// SIMATIC S7-200 project (STEP 7-Micro/WIN), CPU 224 CN REL 02.02

ORGANIZATION_BLOCK 主程序:OB1
TITLE=程序注释
BEGIN
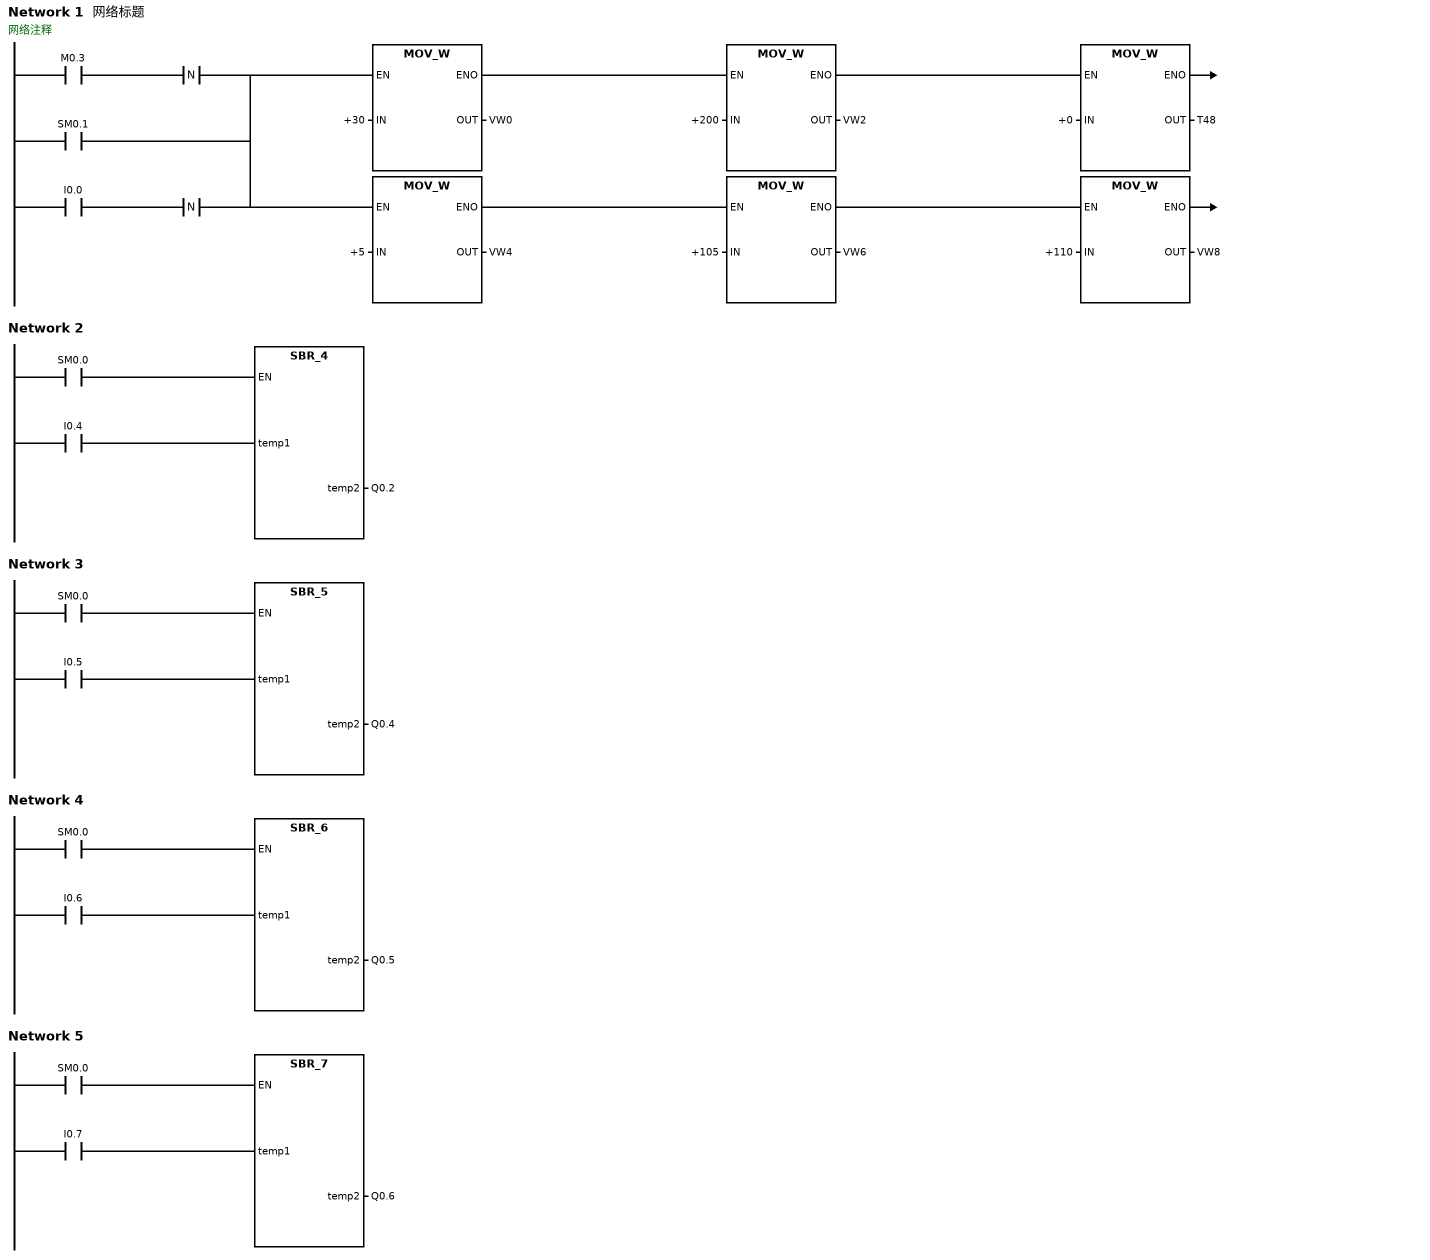
Network 1 // 网络标题
// 网络注释
LD     M0.3
ED
O      SM0.1
LD     I0.0
ED
OLD
LPS
MOVW   +30, VW0
AENO
MOVW   +200, VW2
AENO
MOVW   +0, T48
LPP
MOVW   +5, VW4
AENO
MOVW   +105, VW6
AENO
MOVW   +110, VW8
Network 2
LD     SM0.0
=      L60.0
LD     I0.4
=      L63.7
LD     L60.0
CALL   SBR_4:SBR0, L63.7, Q0.2
Network 3
LD     SM0.0
=      L60.0
LD     I0.5
=      L63.7
LD     L60.0
CALL   SBR_5:SBR1, L63.7, Q0.4
Network 4
LD     SM0.0
=      L60.0
LD     I0.6
=      L63.7
LD     L60.0
CALL   SBR_6:SBR2, L63.7, Q0.5
Network 5
LD     SM0.0
=      L60.0
LD     I0.7
=      L63.7
LD     L60.0
CALL   SBR_7:SBR3, L63.7, Q0.6
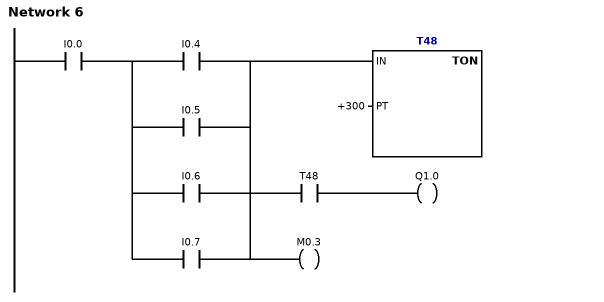
Network 6
// (network saved uncompiled; LAD cells follow)
// row 0: c0 -| |- I0.0 v  c1 -| |- I0.4 v  c2 --  c3 [TON T48 IN:=power@row0, PT:=+300]
// row 1: c0 ^v  c1 -| |- I0.5 ^v  c3 [box]
// row 2: c0 ^v  c1 -| |- I0.6 ^v  c2 -| |- T48  c3 -( ) Q1.0
// row 3: c0 ^  c1 -| |- I0.7 ^  c2 -( ) M0.3
END_ORGANIZATION_BLOCK

SUBROUTINE_BLOCK SBR_4:SBR0
TITLE=子程序注释
VAR_INPUT
temp1:BOOL;	// L0.0 
END_VAR
VAR_OUTPUT
temp2:BOOL;	// L0.1 
END_VAR
BEGIN
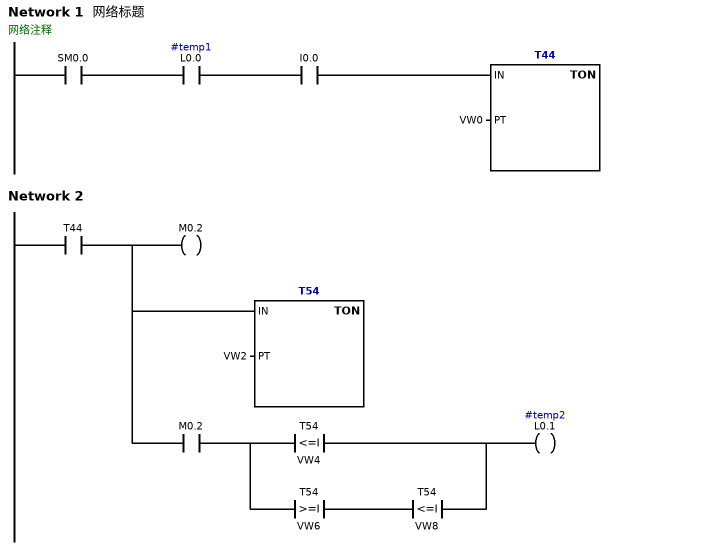
Network 1 // 网络标题
// 网络注释
LD     SM0.0
A      #temp1:L0.0
A      I0.0
TON    T44, VW0
Network 2
LD     T44
=      M0.2
TON    T54, VW2
A      M0.2
LDW<=  T54, VW4
LDW>=  T54, VW6
AW<=   T54, VW8
OLD
ALD
=      #temp2:L0.1
END_SUBROUTINE_BLOCK

SUBROUTINE_BLOCK SBR_5:SBR1
TITLE=
VAR_INPUT
temp1:BOOL;	// L0.0 
END_VAR
VAR_OUTPUT
temp2:BOOL;	// L0.1 
END_VAR
BEGIN
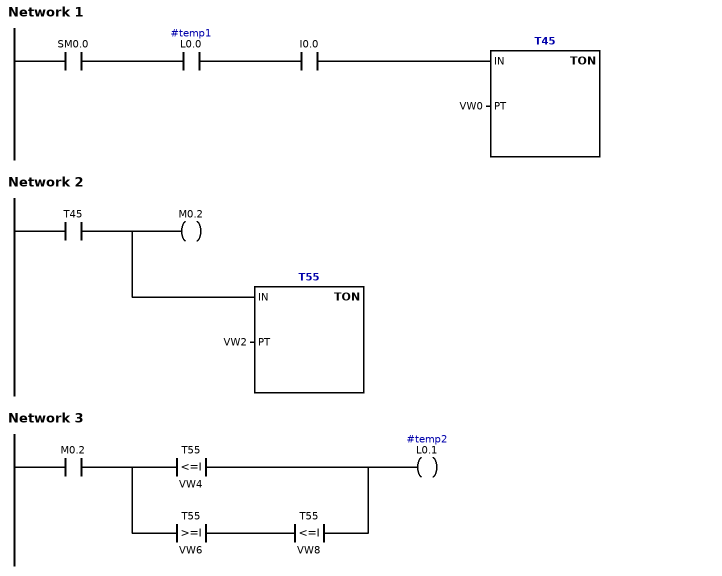
Network 1
LD     SM0.0
A      #temp1:L0.0
A      I0.0
TON    T45, VW0
Network 2
LD     T45
=      M0.2
TON    T55, VW2
Network 3
LD     M0.2
LDW<=  T55, VW4
LDW>=  T55, VW6
AW<=   T55, VW8
OLD
ALD
=      #temp2:L0.1
END_SUBROUTINE_BLOCK

SUBROUTINE_BLOCK SBR_6:SBR2
TITLE=
VAR_INPUT
temp1:BOOL;	// L0.0 
END_VAR
VAR_OUTPUT
temp2:BOOL;	// L0.1 
END_VAR
BEGIN
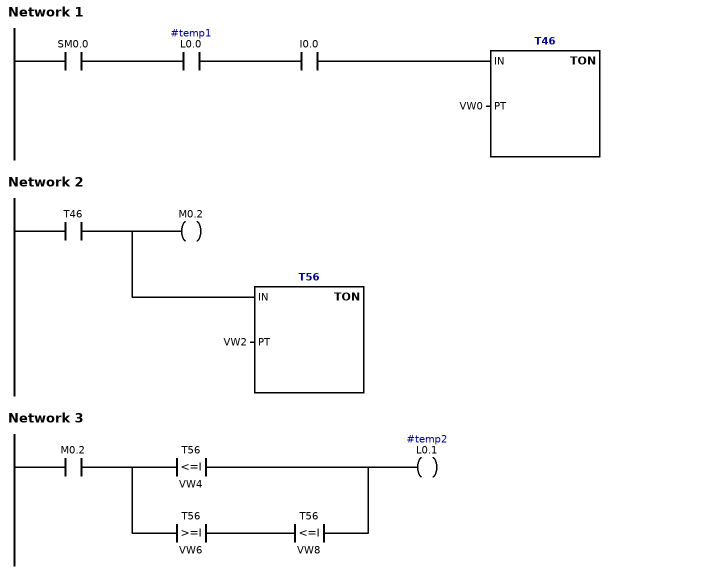
Network 1
LD     SM0.0
A      #temp1:L0.0
A      I0.0
TON    T46, VW0
Network 2
LD     T46
=      M0.2
TON    T56, VW2
Network 3
LD     M0.2
LDW<=  T56, VW4
LDW>=  T56, VW6
AW<=   T56, VW8
OLD
ALD
=      #temp2:L0.1
END_SUBROUTINE_BLOCK

SUBROUTINE_BLOCK SBR_7:SBR3
TITLE=
VAR_INPUT
temp1:BOOL;	// L0.0 
END_VAR
VAR_OUTPUT
temp2:BOOL;	// L0.1 
END_VAR
BEGIN
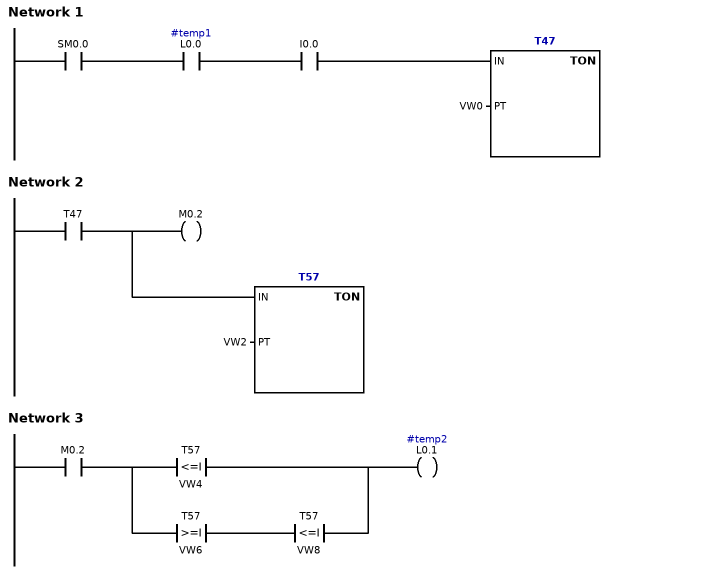
Network 1
LD     SM0.0
A      #temp1:L0.0
A      I0.0
TON    T47, VW0
Network 2
LD     T47
=      M0.2
TON    T57, VW2
Network 3
LD     M0.2
LDW<=  T57, VW4
LDW>=  T57, VW6
AW<=   T57, VW8
OLD
ALD
=      #temp2:L0.1
END_SUBROUTINE_BLOCK
